TYPE ST_ConfigCommon :
STRUCT
END_STRUCT
END_TYPE

(* stored: Version 1.1.0.1, ProductVersion 3.1.4024.12
   DUT ST_ConfigCommon: Id {651c511b-2650-4802-b4ca-9c126ac83ab0} *)
